TYPE T_PointerTest :
STRUCT
	bolPrintOk: BOOL;
	lreActTrayPos_mm : LREAL;
	eState: E_Test;	
END_STRUCT
END_TYPE

(* stored: Version 1.1.0.1, ProductVersion 3.1.0.26
   DUT T_PointerTest: Id {01e8530e-46c9-471b-b78b-6c8a303c30f5} *)
